FUNCTION_BLOCK WaterDischargeOCSLB (* CAT Function Block Type *)
  (* Standard: 61499-2 *)
  (* Version 1.1, 9/30/2026, Claude/Hidryco, Schneider Electric, Rev1.1 - Bomba disponivel = Ready OU Running; Rev1 - Valvula disponivel = Ready OU Aberta *)
  PACKAGE SE.Nereda;
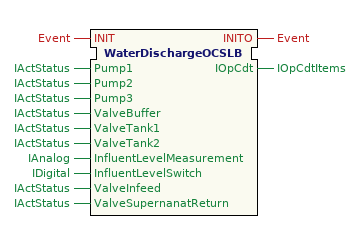
  EVENT_INPUT
    INIT;
  END_EVENT
  EVENT_OUTPUT
    INITO;
  END_EVENT
  SOCKETS
    Pump1 : IActStatus;
    Pump2 : IActStatus;
    Pump3 : IActStatus;
    ValveBuffer : IActStatus;
    ValveTank1 : IActStatus;
    ValveTank2 : IActStatus;
    InfluentLevelMeasurement : IAnalog;
    InfluentLevelSwitch : IDigital;
    ValveInfeed : IActStatus;
    ValveSupernanatReturn : IActStatus;
  END_SOCKETS
  PLUGS
    IOpCdt : IOpCdtItems;
  END_PLUGS
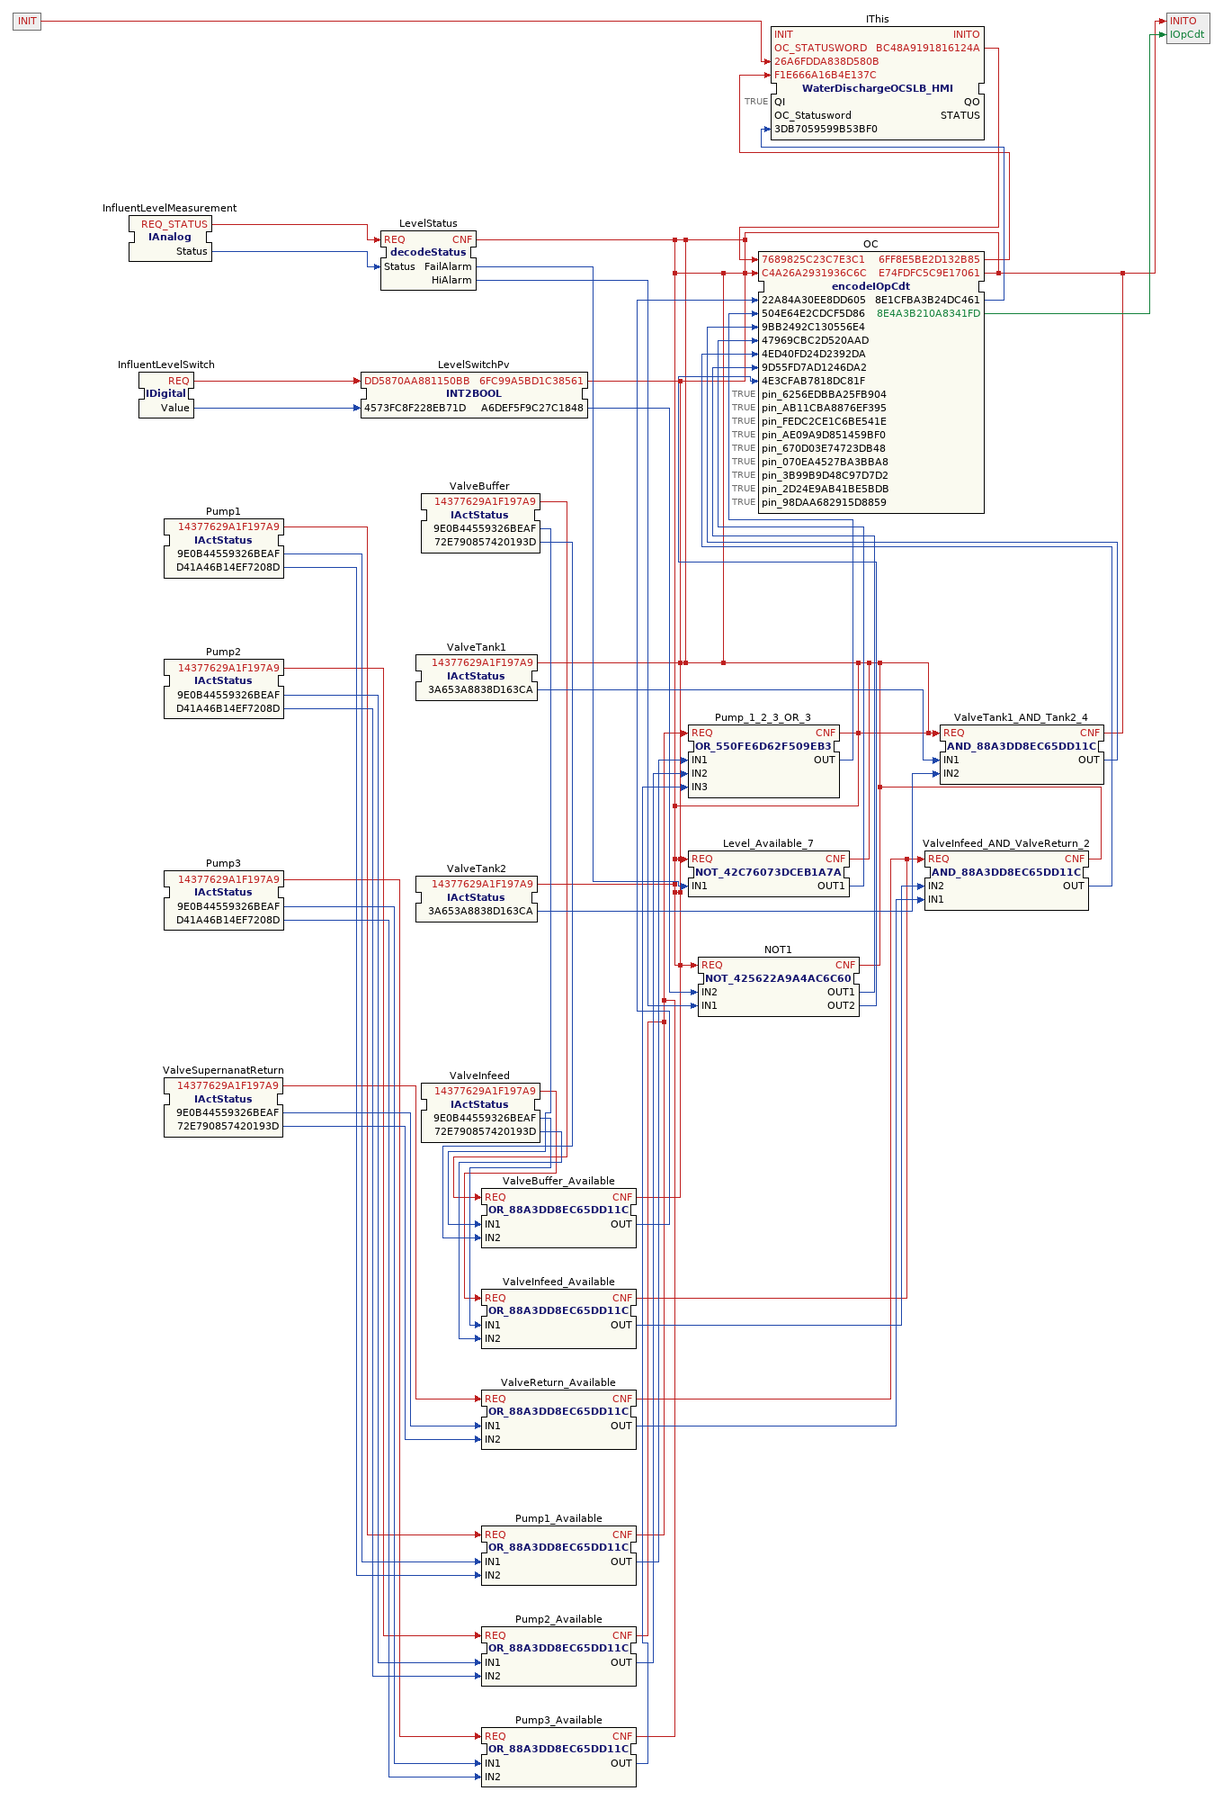
  (* 01 - FUNCTIONNAL INPUT INTERFACE *)
  (* 00 - INITIALIZATION *)
  (* 05 - LOGIC *)
  (* 06 - HMI INTERFACE *)
  (* 03 - FIELD INTERFACE *)
  (* 02 - FUNCTIONNAL OUTPUT INTERFACE *)
  (* Operating Condition Status *)
  (* Operating conditions : 1. Valve Buffer is available 2. Valve Infeed and Valve Return is available 3. Pump 1 or 2 or 3 is available 4. Valve Tank1 AND Tank2 are closed 5. No High level in the influent buffer Level 6. No HH-level in the influent buffer Level Switch 7. Level measurement Level available *)
  FBS
    OC : encodeIOpCdt(pin_6256EDBBA25FB904 := TRUE, pin_AB11CBA8876EF395 := TRUE, pin_FEDC2CE1C6BE541E := TRUE, pin_AE09A9D851459BF0 := TRUE, pin_670D03E74723DB48 := TRUE, pin_070EA4527BA3BBA8 := TRUE, pin_3B99B9D48C97D7D2 := TRUE, pin_2D24E9AB41BE5BDB := TRUE, pin_98DAA682915D8859 := TRUE); (* You set the operating conditions. For the inputs that are not used set a constant to TRUE. *)
    IThis : WaterDischargeOCSLB_HMI(QI := TRUE);
    Pump_1_2_3_OR_3 : OR_550FE6D62F509EB3; {SET_ATTRIBUTE(Configuration.GenericFBType.InterfaceParams, Runtime.Standard#CNT:=3;OUT:BOOL)}
    ValveTank1_AND_Tank2_4 : AND_88A3DD8EC65DD11C; {SET_ATTRIBUTE(Configuration.GenericFBType.InterfaceParams, Runtime.Standard#CNT:=2;OUT:BOOL)}
    Level_Available_7 : NOT_42C76073DCEB1A7A; {SET_ATTRIBUTE(Configuration.GenericFBType.InterfaceParams, Runtime.Standard#CNT:=1;OUT${CNT$}:BOOL)}
    LevelStatus : decodeStatus; {SET_ATTRIBUTE(Configuration.Component.HideUnusedPorts, )}
    LevelSwitchPv : INT2BOOL;
    NOT1 : NOT_425622A9A4AC6C60; {SET_ATTRIBUTE(Configuration.GenericFBType.InterfaceParams, Runtime.Standard#CNT:=2;OUT${CNT$}:BOOL,BOOL)}
    ValveInfeed_AND_ValveReturn_2 : AND_88A3DD8EC65DD11C; {SET_ATTRIBUTE(Configuration.GenericFBType.InterfaceParams, Runtime.Standard#CNT:=2;OUT:BOOL)}
    ValveBuffer_Available : OR_88A3DD8EC65DD11C; {SET_ATTRIBUTE(Configuration.GenericFBType.InterfaceParams, Runtime.Standard#CNT:=2;OUT:BOOL)}
    ValveInfeed_Available : OR_88A3DD8EC65DD11C; {SET_ATTRIBUTE(Configuration.GenericFBType.InterfaceParams, Runtime.Standard#CNT:=2;OUT:BOOL)}
    ValveReturn_Available : OR_88A3DD8EC65DD11C; {SET_ATTRIBUTE(Configuration.GenericFBType.InterfaceParams, Runtime.Standard#CNT:=2;OUT:BOOL)}
    Pump1_Available : OR_88A3DD8EC65DD11C; {SET_ATTRIBUTE(Configuration.GenericFBType.InterfaceParams, Runtime.Standard#CNT:=2;OUT:BOOL)}
    Pump2_Available : OR_88A3DD8EC65DD11C; {SET_ATTRIBUTE(Configuration.GenericFBType.InterfaceParams, Runtime.Standard#CNT:=2;OUT:BOOL)}
    Pump3_Available : OR_88A3DD8EC65DD11C; {SET_ATTRIBUTE(Configuration.GenericFBType.InterfaceParams, Runtime.Standard#CNT:=2;OUT:BOOL)}
  END_FBS
  EVENT_CONNECTIONS
    INIT TO IThis.26A6FDDA838D580B;
    OC.6FF8E5BE2D132B85 TO IThis.F1E666A16B4E137C;
    IThis.BC48A9191816124A TO OC.7689825C23C7E3C1;
    OC.E74FDFC5C9E17061 TO OC.C4A26A2931936C6C;
    OC.E74FDFC5C9E17061 TO INITO;
    ValveBuffer.14377629A1F197A9 TO ValveBuffer_Available.REQ;
    Pump1.14377629A1F197A9 TO Pump1_Available.REQ;
    Pump2.14377629A1F197A9 TO Pump2_Available.REQ;
    Pump3.14377629A1F197A9 TO Pump3_Available.REQ;
    Pump_1_2_3_OR_3.CNF TO OC.C4A26A2931936C6C;
    ValveTank1.14377629A1F197A9 TO ValveTank1_AND_Tank2_4.REQ;
    ValveTank2.14377629A1F197A9 TO ValveTank1_AND_Tank2_4.REQ;
    InfluentLevelMeasurement.REQ_STATUS TO LevelStatus.REQ;
    InfluentLevelSwitch.REQ TO LevelSwitchPv.DD5870AA881150BB;
    LevelStatus.CNF TO OC.C4A26A2931936C6C;
    LevelSwitchPv.6FC99A5BD1C38561 TO OC.C4A26A2931936C6C;
    ValveTank1_AND_Tank2_4.CNF TO OC.C4A26A2931936C6C;
    Level_Available_7.CNF TO OC.C4A26A2931936C6C;
    LevelStatus.CNF TO Level_Available_7.REQ;
    ValveTank2.14377629A1F197A9 TO OC.C4A26A2931936C6C;
    ValveInfeed_AND_ValveReturn_2.CNF TO OC.C4A26A2931936C6C;
    LevelStatus.CNF TO NOT1.REQ;
    NOT1.CNF TO OC.C4A26A2931936C6C;
    LevelSwitchPv.6FC99A5BD1C38561 TO NOT1.REQ;
    ValveInfeed.14377629A1F197A9 TO ValveInfeed_Available.REQ;
    ValveSupernanatReturn.14377629A1F197A9 TO ValveReturn_Available.REQ;
    ValveBuffer_Available.CNF TO OC.C4A26A2931936C6C;
    ValveInfeed_Available.CNF TO ValveInfeed_AND_ValveReturn_2.REQ;
    ValveReturn_Available.CNF TO ValveInfeed_AND_ValveReturn_2.REQ;
    Pump1_Available.CNF TO Pump_1_2_3_OR_3.REQ;
    Pump2_Available.CNF TO Pump_1_2_3_OR_3.REQ;
    Pump3_Available.CNF TO Pump_1_2_3_OR_3.REQ;
  END_CONNECTIONS
  DATA_CONNECTIONS
    OC.8E1CFBA3B24DC461 TO IThis.3DB7059599B53BF0;
    ValveBuffer_Available.OUT TO OC.22A84A30EE8DD605;
    Pump1_Available.OUT TO Pump_1_2_3_OR_3.IN1;
    Pump2_Available.OUT TO Pump_1_2_3_OR_3.IN2;
    Pump3_Available.OUT TO Pump_1_2_3_OR_3.IN3;
    Pump_1_2_3_OR_3.OUT TO OC.504E64E2CDCF5D86;
    ValveTank1.3A653A8838D163CA TO ValveTank1_AND_Tank2_4.IN1;
    ValveTank2.3A653A8838D163CA TO ValveTank1_AND_Tank2_4.IN2;
    ValveTank1_AND_Tank2_4.OUT TO OC.9BB2492C130556E4;
    InfluentLevelMeasurement.Status TO LevelStatus.Status;
    InfluentLevelSwitch.Value TO LevelSwitchPv.4573FC8F228EB71D;
    LevelSwitchPv.A6DEF5F9C27C1848 TO NOT1.IN2;
    LevelStatus.FailAlarm TO Level_Available_7.IN1;
    Level_Available_7.OUT1 TO OC.47969CBC2D520AAD;
    ValveInfeed_AND_ValveReturn_2.OUT TO OC.4ED40FD24D2392DA;
    LevelStatus.HiAlarm TO NOT1.IN1;
    NOT1.OUT1 TO OC.9D55FD7AD1246DA2;
    NOT1.OUT2 TO OC.4E3CFAB7818DC81F;
    ValveInfeed_Available.OUT TO ValveInfeed_AND_ValveReturn_2.IN2;
    ValveReturn_Available.OUT TO ValveInfeed_AND_ValveReturn_2.IN1;
    ValveBuffer.9E0B44559326BEAF TO ValveBuffer_Available.IN1;
    ValveBuffer.72E790857420193D TO ValveBuffer_Available.IN2;
    ValveInfeed.9E0B44559326BEAF TO ValveInfeed_Available.IN1;
    ValveInfeed.72E790857420193D TO ValveInfeed_Available.IN2;
    ValveSupernanatReturn.9E0B44559326BEAF TO ValveReturn_Available.IN1;
    ValveSupernanatReturn.72E790857420193D TO ValveReturn_Available.IN2;
    Pump1.9E0B44559326BEAF TO Pump1_Available.IN1;
    Pump1.D41A46B14EF7208D TO Pump1_Available.IN2;
    Pump2.9E0B44559326BEAF TO Pump2_Available.IN1;
    Pump2.D41A46B14EF7208D TO Pump2_Available.IN2;
    Pump3.9E0B44559326BEAF TO Pump3_Available.IN1;
    Pump3.D41A46B14EF7208D TO Pump3_Available.IN2;
  END_CONNECTIONS
  ADAPTER_CONNECTIONS
    OC.8E4A3B210A8341FD TO IOpCdt;
  END_CONNECTIONS
END_FUNCTION_BLOCK
